// TIA Portal V19 export
FUNCTION_BLOCK "TYPIC_C701_IF_VAT"   // FB69, FBD
TITLE = TYPIC_C701_IF_VAT: Expansievaten
{ S7_Optimized_Access := 'TRUE' }
AUTHOR : OCOTECH
FAMILY : Typical
NAME : C701.713
// Logisch Object Besturing: C701.713
// 
// De interne functie Expansievaten verzorgt de bewaking van een expansievat behorend tot de klimaatinstallatie.
// In zowel de collector verwarming als koeling is er een expansievat.
// stored: MemoryReserve 10, SetENOAutomatically false
   VAR_INPUT
      IN_AL_VE { ExternalAccessible := 'False'; ExternalVisible := 'False'; ExternalWritable := 'False'} : Bool;   // Alarm lage druk expansievat verwarming (1 = Alarm)
      IN_DME_VE { ExternalAccessible := 'False'; ExternalVisible := 'False'; ExternalWritable := 'False'} : Real;   // Drukmeting expansievat verwarming
      IN_AL_KO { ExternalAccessible := 'False'; ExternalVisible := 'False'; ExternalWritable := 'False'} : Bool;   // Alarm lage druk expansievat koeling (1 = Alarm)
      IN_DME_KO { ExternalAccessible := 'False'; ExternalVisible := 'False'; ExternalWritable := 'False'} : Real;   // Drukmeting expansievat koeling
   END_VAR
   VAR_OUTPUT
      VAR_IF_VAT { ExternalAccessible := 'False'; ExternalVisible := 'False'; ExternalWritable := 'False'} : "C701_VAR_IF_VAT_TYPIC";   // Struct met alle variabelen naar bovenliggende functies
   END_VAR
   VAR
      STO { ExternalWritable := 'False'} : Struct   // Storingen
         A001 : Bool;   // Alarm lage druk expansievat verwarming
         A002 : Bool;   // Fout drukmeting expansievat verwarming
         A003 : Bool;   // Alarm lage druk expansievat koeling
         A004 : Bool;   // Fout drukmeting expansievat koeling
      END_STRUCT;
      VAR { ExternalWritable := 'False'} : Struct   // Variabelen
         DME_VE : Real;   // Drukmeting expansievat verwarming
         DME_KO : Real;   // Drukmeting expansievat koeling
      END_STRUCT;
   END_VAR
BEGIN

REGION Network 1: START
END_REGION

REGION Network 2: +++ Metingen +++
   // inlezen van drukmeting.
END_REGION

REGION Network 3: +++ Storingen en meldingen +++
   // aanmaken van storingen en meldingen.
END_REGION

REGION Network 4: Storing A001: Alarm lage druk expansievat verwarming
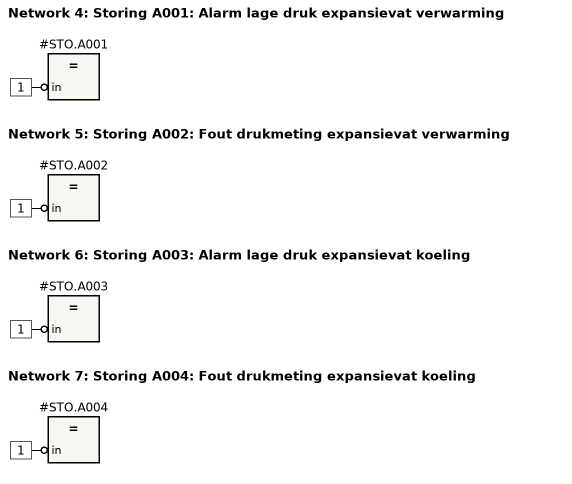
   #STO.A001 := NOT 1;
END_REGION

REGION Network 5: Storing A002: Fout drukmeting expansievat verwarming
   #STO.A002 := NOT 1;
END_REGION

REGION Network 6: Storing A003: Alarm lage druk expansievat koeling
   #STO.A003 := NOT 1;
END_REGION

REGION Network 7: Storing A004: Fout drukmeting expansievat koeling
   #STO.A004 := NOT 1;
END_REGION

REGION Network 8 (SCL): EINDE
   // Variabelen van intern scada rakvlak naar outputs copieren
   #VAR_IF_VAT.STO := #STO;
END_REGION
END_FUNCTION_BLOCK
